// TIA Portal V16 export
// export: Created 2023-11-14T19:43:18.8284471Z, ExportSetting WithDefaults, DisplayName Totally Integrated Automation Portal, DisplayVersion V16, DisplayName TIA Portal Version Control Interface, DisplayVersion V16, DisplayName TIA Portal Openness, DisplayVersion V16, DisplayName SINAMICS Startdrive Advanced, DisplayVersion V16, DisplayName SINAMICS Startdrive G130, G150, S120, S150, SINAMICS MV, S210, DisplayVersion V16, DisplayName SINAMICS Startdrive G110M, G120, G120C, G120D, G120P, DisplayVersion V16, DisplayName STEP 7 Professional, DisplayVersion V16, DisplayName STEP 7 Safety, DisplayVersion V16, DisplayName WinCC Professional, DisplayVersion V16
DATA_BLOCK "Prom_FilterV2_DB"   // DB25
VERSION : 0.1
// stored: AutoNumber true, DBAccessibleFromOPCUA true, InstanceOfName Prom_FilterV2, InstanceOfType FB
"Prom_FilterV2"
   // VAR_INPUT
   //    Scale_Value { ExternalAccessible := 'False'; ExternalVisible := 'False'; ExternalWritable := 'False'} : Real;
   //    Inf_Limit { ExternalAccessible := 'False'; ExternalVisible := 'False'; ExternalWritable := 'False'} : Real;
   //    Sup_Limit { ExternalAccessible := 'False'; ExternalVisible := 'False'; ExternalWritable := 'False'} : Real;
   //    Cal { ExternalAccessible := 'False'; ExternalVisible := 'False'; ExternalWritable := 'False'} : Real;
   //    Filter_Set_Time : Time;
   //    Max_Analog_Value : UInt;
   // END_VAR
   // VAR_OUTPUT
   //    Prom_Filter : Real;
   // END_VAR
   // VAR
   //    i { ExternalVisible := 'False'} : Int;
   // END_VAR
   // VAR RETAIN
   //    i_Acum { ExternalVisible := 'False'} : Real;
   // END_VAR
   // VAR
   //    Pv_Value : Real;
   //    Pv_Aux1 : Real;
   //    En_Filter_Timer : Bool;
   //    Filter_P_Time : Time;
   //    Filter_TImer { S7_SetPoint := 'True'} : TONR_TIME;
   // END_VAR
BEGIN
END_DATA_BLOCK
